{attribute 'qualified_only'}
{attribute 'strict'}
TYPE EterCAT_State :
(
	INIT,
	PREOP,
	BOOT,
	SAFEOP,
	OP,
	Signals_Error,
	Invalid_VendorID,
	Disabeld,
	Not_Present,
	Signgals_Link_error,
	Signals_unexpected_Link
);
END_TYPE

(* stored: Version 1.1.0.1, ProductVersion 3.1.4024.10
   DUT EterCAT_State: Id {2c83d28b-ef82-4212-a608-9e7de67598b3} *)
